Staubli VAL3: refreshStatic.pgx

program refreshStatic()
  local string l_sMenu
begin
  cls()
  //
  // set the view of the page..
  //
  // SET THE PAGE NUMBER
  use:nPage=100
  // USE <>PROFILE for <>PAGE
  use:nPage=use:nPage+abs(limit(saveData:mode,0,2)-2)
  // SET THE VIEW OF THE PAGE
  call language2:page(l_sMenu,use:nPage)
  // define the menu
  call use:stringToArray(l_sMenu,sMenu)
  //
  call use:setMenu(sMenu,true,3)
  call use:getMenu(sMenu,bButton)
  //
  // CREATE THE LIST
  //
  // define your list size for default
  call use:setSizeList(19,0,19,11)
  call use:setView(bLarge)
  //
  call use:listcreate("")
  //
end
